(* IEC 61131-3 sources: CodesysTest/alpha/export/FBs/Fault/FB_Fault.pou/Passive Properties/PassiveExitConeyorOverride.prop, 1 file *)

(* ---- Get.pm.st ---- *)
(*#-#-#-#-#-#-#-#-#-#---Declaration---#-#-#-#-#-#-#-#-#-#-#-#-#*)

VAR
END_VAR
(*#-#-#-#-#-#-#-#-#-#---Implementation---#-#-#-#-#-#-#-#-#-#-#-#-#*)

PassiveExitConeyorOverride := _exitConveyorOverride;
